FUNCTION FC_MeanOfArray : REAL
VAR_INPUT CONSTANT
	n 		: INT;
	aArray 	: ARRAY [1..n] OF REAL;
END_VAR
VAR
	i 		: INT;
	fTemp 	: REAL	:= 0;
END_VAR

FOR i := 1 TO n DO
	fTemp := fTemp + aArray[i];
END_FOR

FC_MeanOfArray := fTemp / n;

END_FUNCTION

(* stored: Version 1.1.0.1, ProductVersion 3.1.4024.0
   POU FC_MeanOfArray: Id {f0241d9d-3185-4cdb-ac24-bed62ae8bcca}, SpecialFunc None *)
